Yaskawa INFORM job: SKRZYNIA_4640_0_STOPNI_1OBR.JBI

/JOB
//NAME SKRZYNIA_4640_0_STOPNI_1OBR
///FOLDERNAME 02-SKRZYNIE_JOBS
//POS
///NPOS 503,503,0,43,0,0
///TOOL 0
///POSTYPE PULSE
///PULSE
C00000=1055,-24125,84372,288,19725,204
C00001=1055,-24125,84372,288,19725,204
C00002=0,-15438,65714,0,-68532,0
C00003=25524,-25821,36823,19654,-58495,38520
C00004=23988,-24960,37134,18595,-57837,38812
C00005=22822,-23954,37534,17811,-57199,39017
C00006=22935,-24057,37491,17887,-57262,38997
C00007=20006,-24258,37408,15644,-56932,39751
C00008=24402,-25289,37013,18874,-58060,38740
C00009=22585,-24665,40358,17164,-59622,30036
C00010=23477,-23257,40205,18030,-58646,29630
C00011=22519,-22398,40568,17384,-58125,29795
C00012=22700,-22567,40495,17506,-58225,29764
C00013=19339,-22794,40398,14955,-57865,30607
C00014=24825,-24328,39798,18931,-59350,29401
C00015=25524,-25821,36823,19654,-58495,38520
C00016=23988,-24960,37134,18595,-57837,38812
C00017=22822,-23954,37534,17811,-57199,39017
C00018=22935,-24057,37491,17887,-57262,38997
C00019=20006,-24258,37408,15644,-56932,39751
C00020=24402,-25289,37013,18874,-58060,38740
C00021=22585,-24665,40358,17164,-59622,30036
C00022=23477,-23257,40205,18030,-58646,29630
C00023=22519,-22398,40568,17384,-58125,29795
C00024=22700,-22567,40495,17506,-58225,29764
C00025=19339,-22794,40398,14955,-57865,30607
C00026=24825,-24328,39798,18931,-59350,29401
C00027=32755,-32613,25711,29640,-48730,33694
C00028=25632,-30899,26166,23992,-46203,35378
C00029=24264,-29862,26497,22996,-45413,35639
C00030=24403,-29974,26459,23097,-45496,35612
C00031=20575,-30233,26374,19602,-44891,36810
C00032=26556,-31526,25988,24663,-46720,35206
C00033=31152,-34007,25432,27964,-49085,34371
C00034=14779,-22420,82153,5620,-31515,42478
C00035=14779,-22420,82153,5620,-31515,42478
C00036=27667,-31817,30876,40298,-29340,25942
C00037=30467,-34548,18624,42252,-31099,25545
C00038=27667,-31817,21023,40298,-29340,25942
C00039=26226,-30681,21430,39338,-28403,26129
C00040=26403,-30829,21375,39455,-28520,26106
C00041=23300,-31093,21277,35654,-27590,27434
C00042=27667,-31817,21023,40298,-29340,25942
C00043=33767,-35384,20030,44426,-32984,25136
C00044=17528,-33021,25719,14295,-44761,40001
C00045=28412,-21339,35361,20830,-70681,36412
C00046=27333,-20260,35973,20228,-70115,36596
C00047=27560,-20497,35837,20355,-70235,36556
C00048=24830,-20816,35654,18694,-69859,37222
C00049=28877,-18893,40191,20941,-72149,36569
C00050=27817,-32566,25782,25532,-47502,36865
C00051=25779,-31294,26110,24054,-46400,37243
C00052=24344,-30243,26427,23007,-45578,37515
C00053=24432,-30312,26405,23072,-45630,37498
C00054=20021,-30599,26315,19050,-44944,38872
C00055=26262,-31616,26021,24405,-46667,37153
C00056=27439,-32346,25835,25259,-47302,36935
C00057=25659,-31170,26146,23974,-46312,37260
C00058=24581,-30384,26384,23190,-45695,37464
C00059=24689,-30466,26358,23269,-45758,37444
C00060=20001,-30771,26264,18999,-45026,38899
C00061=26308,-31607,26026,24448,-46671,37139
C00062=26309,-31604,29506,24448,-46670,37138
C00063=58801,-24999,56179,43319,-3155,35712
C00064=58801,-24999,56179,43319,-3155,35712
C00065=58801,-24999,56179,43319,-54497,35712
C00066=29920,-29398,24569,49034,-27892,27689
C00067=29115,-28721,24834,48649,-27358,27707
C00068=27674,-27540,25333,47889,-26423,27783
C00069=27794,-27645,25287,47952,-26502,27777
C00070=24751,-27949,25156,44290,-25406,29014
C00071=29115,-28721,24834,48649,-27358,27707
C00072=40370,-34602,23054,55084,-33911,26929
C00073=27585,-47842,-289,32095,-40789,28095
C00074=4801,-35772,25187,4593,-28023,-82032
C00075=17634,-23800,39238,9573,-31425,-73339
C00076=17634,-23800,39238,9573,-31425,-73339
C00077=16549,-22464,39800,8390,-30730,-72975
C00078=16684,-22641,39722,8536,-30818,-73021
C00079=16684,-19968,45512,8078,-32771,-72767
C00080=17634,-23800,39238,9573,-31425,-73339
C00081=17837,-21535,44509,9322,-33342,-73155
C00082=17837,-21535,44509,9322,-33342,-73155
C00083=16866,-20378,45014,8305,-32755,-72853
C00084=17032,-20588,44918,8481,-32857,-72905
C00085=17032,-17542,51480,8009,-35060,-72636
C00086=17837,-21535,44509,9322,-33342,-73155
C00087=-20829,-18800,50532,-12466,-37179,-77446
C00088=-19934,-17904,50946,-11618,-36715,-77676
C00089=-20044,-18019,50891,-11723,-36773,-77647
C00090=-20044,-15288,56753,-11218,-38713,-77950
C00091=-20966,-18928,50473,-12596,-37250,-77413
C00092=-20884,-26676,33664,-14451,-31668,-76336
C00093=-20884,-26676,33664,-14451,-31668,-76336
C00094=-19557,-25338,34176,-13080,-30873,-76751
C00095=-19691,-25483,34117,-13220,-30955,-76709
C00096=-19691,-22773,39998,-12506,-32911,-77106
C00097=-20642,-26447,33747,-14206,-31526,-76411
C00098=-33629,-40566,17444,-29603,-33447,-71192
C00099=-33629,-40566,17444,42578,-32312,-84654
C00100=-42160,-31266,16400,42578,-32312,-84654
C00101=-87798,-804,48829,-20188,-26072,-60966
C00102=-76454,-11934,10236,-25964,7954,-64922
C00103=-76448,-11928,10235,-25961,7944,-64914
C00104=-68643,-7759,-23318,-14097,50582,-74897
C00105=-70868,-8793,-8075,-29663,30364,-70765
C00106=-67243,-1968,12282,-49553,26687,-63567
C00107=-68655,-309,14069,-48513,25966,-64203
C00108=-67497,-1678,12591,-49367,26558,-63682
C00109=-71436,-723,2905,-26484,35140,-73726
C00110=-71436,176,6426,-27636,33595,-73066
C00111=-71434,778,8668,-28412,32633,-72624
C00112=-68624,-2689,-85,-28291,36551,-72622
C00113=-99375,3692,5712,40719,48607,-84097
C00114=-94964,4957,10918,40408,44640,-83792
C00115=-93063,6047,12199,39572,43744,-83178
C00116=-94964,4957,10918,40408,44640,-83792
C00117=-94964,5754,13918,41385,43553,-84439
C00118=-94964,4957,10918,40408,44640,-83792
C00119=-90271,-412,-5146,23417,46876,-76529
C00120=-83133,-4088,-8267,6704,41492,-71542
C00121=-83133,-4088,-8267,6704,41492,-71542
C00122=-83133,-4088,-8267,6704,41492,-11598
C00123=-83133,-16026,-8267,6704,41492,-11598
C00124=-83133,-16026,-8267,6704,41492,-11598
C00125=-48225,-19387,30619,3889,32460,-6728
C00126=56943,-39861,25115,1795,-37402,-69601
C00127=29960,-38386,-19607,-115769,-41858,-24264
C00128=65721,-6478,18155,-133323,-22195,3361
C00129=70544,4411,32968,-134868,-18623,4660
C00130=71874,8263,38598,-134556,-17327,4659
C00131=72629,9390,40002,-135279,-16924,5107
C00132=71441,7638,37831,-134139,-17555,4406
C00133=77146,8888,25050,-166574,-32612,18372
C00134=77146,10029,28643,-166204,-31014,18167
C00135=77146,11198,32202,-165803,-29459,17947
C00136=75508,4678,16951,-165715,-35157,17778
C00137=68680,12216,24468,-164340,-40455,-13359
C00138=68362,12845,25743,-164045,-40097,-13561
C00139=68362,13700,28585,-163752,-38808,-13742
C00140=68362,12845,25743,-164045,-40097,-13561
C00141=64993,-1168,28876,-102971,-10760,-49875
C00142=63888,481,30670,-102324,-11438,-50313
C00143=64993,-1168,28876,-102971,-10760,-49875
C00144=58588,-14653,4620,-120782,-19611,-35794
C00145=29960,-38386,-19607,-115769,-41858,-24264
C00146=56943,-39861,25115,1795,-37402,-69601
C00147=-1002,-39861,25115,1795,-37402,-69601
C00148=-1001,-39858,25114,1795,-37402,0
C00149=6591,-33902,35532,5956,-1761,-1932
C00150=6592,-33900,35531,103508,-35512,-26314
C00151=-99253,-13690,44082,59847,13407,-31313
C00152=-85045,-36869,-4353,28502,-22832,-52282
C00153=-92346,-18713,13565,21110,-22545,-55257
C00154=-85732,-21202,11427,30682,-24763,-59235
C00155=-84559,-15616,15722,33768,-24118,-60665
C00156=-84150,-13282,17685,34842,-23935,-61163
C00157=-83260,-12880,18034,36130,-24218,-61709
C00158=-84150,-13282,17685,34842,-23935,-61163
C00159=-85365,-11775,19006,33430,-23307,-60600
C00160=-84150,-13282,17685,34842,-23935,-61163
C00161=-85786,-16909,14677,31743,-23900,-59790
C00162=-84150,-13282,17685,34842,-23935,-61163
C00163=-83215,-12861,18051,36194,-24233,-61735
C00164=-84150,-13282,17685,34842,-23935,-61163
C00165=-85327,-11825,18959,33476,-23327,-60618
C00166=-84150,-13282,17685,34842,-23935,-61163
C00167=-87841,-18519,13420,28367,-23534,-58339
C00168=-84150,-13282,17685,34842,-23935,-61163
C00169=-83292,-12894,18020,36083,-24208,-61688
C00170=-84150,-13282,17685,34842,-23935,-61163
C00171=-85185,-12008,18799,33646,-23400,-60687
C00172=-84150,-13282,17685,34842,-23935,-61163
C00173=-86371,-18277,13606,30568,-23951,-59265
C00174=-84345,-13370,17612,34554,-23873,-61041
C00175=-83240,-12871,18042,36158,-24225,-61720
C00176=-84345,-13370,17612,34554,-23873,-61041
C00177=-85365,-12110,18711,33368,-23345,-60568
C00178=-84345,-13370,17612,34554,-23873,-61041
C00179=-86191,-19647,12567,30467,-24278,-59187
C00180=-84345,-13372,17610,34552,-23873,-61039
C00181=-83096,-12807,18098,36363,-24268,-61804
C00182=-84345,-13372,17610,34552,-23873,-61039
C00183=-85268,-12232,18600,33480,-23393,-60612
C00184=-84345,-13372,17610,34552,-23873,-61039
C00185=-84814,-16043,15376,33312,-24093,-60464
C00186=-84104,-13265,17702,34906,-23948,-61189
C00187=-82960,-12743,18153,36555,-24313,-61887
C00188=-84104,-13265,17702,34906,-23948,-61189
C00189=-84979,-12194,18635,33901,-23496,-60788
C00190=-84104,-13265,17702,34906,-23948,-61189
C00191=-86610,-16845,14732,30573,-23614,-59301
C00192=-84104,-13265,17702,34906,-23948,-61189
C00193=-82793,-12667,18222,36790,-24370,-61986
C00194=-84104,-13265,17702,34906,-23948,-61189
C00195=-84888,-12305,18537,34004,-23540,-60830
C00196=-84104,-13265,17702,34906,-23948,-61189
C00197=-83806,-19585,12613,33764,-25080,-60559
C00198=-83675,-13072,17868,35530,-24083,-61453
C00199=-82553,-12556,18319,37130,-24451,-62127
C00200=-83675,-13072,17868,35530,-24083,-61453
C00201=-84378,-12223,18610,34735,-23716,-61138
C00202=-83675,-13072,17868,35530,-24083,-61453
C00203=-87149,-17993,13826,29513,-23647,-58830
C00204=-84104,-13265,17702,34906,-23948,-61189
C00205=-82640,-12594,18285,37014,-24425,-62079
C00206=-84104,-13265,17702,34906,-23948,-61189
C00207=-84792,-12429,18430,34119,-23592,-60877
C00208=-84104,-13265,17702,34906,-23948,-61189
C00209=-83583,-9185,30892,23668,-36042,-57025
C00210=-85789,-8328,35795,20592,-37093,-55378
C00211=-85786,-16735,14816,31782,-23869,-59812
C00212=-84103,-13263,17702,34906,-23947,-61191
C00213=-83225,-12865,18046,36177,-24227,-61729
C00214=-84103,-13263,17702,34906,-23947,-61191
C00215=-84774,-12447,18412,34138,-23599,-60886
C00216=-84103,-13263,17702,34906,-23947,-61191
C00217=-86149,-16246,6730,18897,-35239,-57128
C00218=-86244,-15289,7532,18875,-35060,-57127
C00219=-85361,-14893,7870,19824,-35193,-57574
C00220=-86244,-15289,7532,18875,-35060,-57127
C00221=-86889,-14409,8282,18264,-34784,-56850
C00222=-86244,-15289,7532,18875,-35060,-57127
C00223=-90262,-21765,2389,14114,-35574,-54847
C00224=-90262,-21765,2389,28730,-17672,-54847
C00225=-89967,-19086,25635,28730,-17672,-54847
C00226=568,-24029,84339,168,19981,112
C00227=568,-24677,83015,164,20405,113
C00228=101153,-24598,83176,165,20353,113
C00229=101153,-24598,83176,165,20353,113
C00230=89967,-19086,25635,-28730,-17672,54847
C00231=90262,-21765,2389,-28730,-17672,54847
C00232=86932,-18662,4771,-17876,-35519,56628
C00233=86578,-15436,7408,-18515,-35011,56957
C00234=85428,-14922,7844,-19753,-35183,57541
C00235=84405,-14447,8250,-20842,-35348,58054
C00236=85428,-14922,7844,-19753,-35183,57541
C00237=86134,-13973,8661,-19091,-34881,57237
C00238=85428,-14922,7844,-19753,-35183,57541
C00239=85786,-16735,14816,-31782,-23869,59812
C00240=83514,-12996,17929,-35760,-24132,61552
C00241=82296,-12429,18424,-37488,-24534,62281
C00242=83514,-12996,17929,-35760,-24132,61552
C00243=84266,-12085,18725,-34910,-23738,61214
C00244=83514,-12996,17929,-35760,-24132,61552
C00245=87323,-6914,39851,-18853,-38149,44508
C00246=83118,-12818,18089,-36330,-24263,61791
C00247=81969,-12276,18566,-37944,-24648,62472
C00248=83118,-12818,18089,-36330,-24263,61791
C00249=83927,-11846,18941,-35423,-23842,61433
C00250=83118,-12818,18089,-36330,-24263,61791
C00251=83806,-19585,12613,-33764,-25080,60559
C00252=83148,-12832,18077,-36287,-24254,61773
C00253=81889,-12236,18598,-38058,-24676,62520
C00254=83148,-12832,18077,-36287,-24254,61773
C00255=83900,-11930,18867,-35446,-23862,61440
C00256=83148,-12832,18077,-36287,-24254,61773
C00257=86610,-16845,14732,-30573,-23614,59301
C00258=82493,-13239,17725,-37070,-24559,62089
C00259=81442,-12739,18159,-38529,-24915,62703
C00260=82493,-13239,17725,-37070,-24559,62089
C00261=83435,-12133,18689,-36040,-24063,61682
C00262=82493,-13239,17725,-37070,-24559,62089
C00263=84814,-16043,15376,-33312,-24093,60464
C00264=82555,-13613,17404,-36910,-24580,62015
C00265=81369,-13053,17885,-38558,-24979,62709
C00266=82555,-13613,17404,-36910,-24580,62015
C00267=83568,-12431,18429,-35805,-24046,61580
C00268=82555,-13613,17404,-36910,-24580,62015
C00269=86191,-19647,12567,-30467,-24278,59187
C00270=82500,-13648,17375,-36975,-24607,62039
C00271=81594,-13224,17740,-38236,-24911,62571
C00272=82500,-13648,17375,-36975,-24607,62039
C00273=83449,-12543,18332,-35941,-24104,61633
C00274=82500,-13648,17375,-36975,-24607,62039
C00275=86371,-18277,13606,-30568,-23951,59265
C00276=82904,-13790,17251,-36416,-24470,61808
C00277=81796,-13275,17692,-37971,-24838,62464
C00278=82904,-13790,17251,-36416,-24470,61808
C00279=83696,-12867,18046,-35547,-24051,61466
C00280=82904,-13790,17251,-36416,-24470,61808
C00281=87841,-18519,13420,-28367,-23534,58339
C00282=82748,-13879,17174,-36603,-24542,61883
C00283=81789,-13434,17554,-37946,-24861,62449
C00284=82748,-13879,17174,-36603,-24542,61883
C00285=83603,-12888,18026,-35668,-24086,61514
C00286=82748,-13879,17174,-36603,-24542,61883
C00287=85786,-16909,14677,-31743,-23900,59790
C00288=82339,-14116,16972,-37087,-24733,62079
C00289=81557,-13752,17280,-38171,-24994,62536
C00290=82339,-14116,16972,-37087,-24733,62079
C00291=83390,-12909,18006,-35951,-24172,61633
C00292=82339,-14116,16972,-37087,-24733,62079
C00293=85732,-21202,11427,-30682,-24763,59235
C00294=82398,-14365,16763,-36952,-24745,62014
C00295=81340,-13876,17176,-38416,-25096,62632
C00296=82398,-14365,16763,-36952,-24745,62014
C00297=83629,-12951,17972,-35620,-24090,61491
C00298=82398,-14365,16763,-36952,-24745,62014
C00299=83775,-36460,5778,-32556,-23750,56951
C00300=69856,-53931,-13446,-33557,-28911,29591
C00301=43695,-41610,22646,45477,-37580,9181
C00302=79833,-32060,29151,65065,-75499,17030
C00303=46589,-23543,32575,47437,-59456,19719
C00304=35046,-28601,21000,31995,-60106,26294
C00305=20995,-31929,9410,15929,-60729,34224
C00306=58029,-25484,23838,55879,-68285,17494
C00307=64424,-28491,31029,58630,-66351,17656
C00308=34280,-39622,35434,31197,-32089,9395
C00309=0,-52280,40443,0,6876,0
C00310=23755,-47704,18289,26329,-25233,13971
C00311=32804,-46073,6525,41905,-31120,14425
C00312=62562,-39100,6547,70046,-55853,12125
C00313=48126,-33841,8393,64372,-47199,12361
C00314=31253,-44096,-7366,36514,-42480,22085
C00315=59828,-44646,-5405,72855,-48572,12139
C00316=0,-38761,66314,0,-763,0
C00317=0,-44757,54667,0,2744,0
C00318=16657,-42063,37160,20008,-15173,6616
C00319=40382,-38226,12225,48505,-40693,16039
C00320=55481,-27484,23768,62968,-54833,11978
C00321=49931,-26522,24223,59987,-51967,12537
C00322=41382,-34078,10932,46059,-50502,16311
C00323=55330,-33748,11238,57660,-59334,12681
C00324=57521,-31202,17284,65112,-55174,10876
C00325=49952,-26929,23567,59763,-52208,12588
C00326=49645,-31441,12217,55064,-56016,13120
C00327=55330,-33748,11238,57660,-59334,12681
C00328=78664,-24436,10378,82837,-79111,12029
C00329=75189,-23065,11287,81851,-76948,11927
C00330=75189,-45249,11287,81851,-38847,11927
C00331=39199,-45249,11287,81851,-83130,11927
C00332=39199,-45249,11287,81851,-83130,11927
C00333=0,-24026,84338,1,19977,2
C00334=0,-24026,84338,1,19977,2
C00335=4264,-34194,25387,4006,-26954,-29436
C00336=4264,-34194,25387,4006,-26954,-81856
C00337=-21478,-27798,32214,-15234,-31599,-76056
C00338=-19679,-23059,39354,-12567,-32689,-77067
C00339=16724,-20576,44291,8212,-32395,-72836
C00340=21329,-26386,39716,13285,-34016,-74401
C00341=-23778,-26243,38799,-16502,-35132,-75964
C00342=-20075,-15782,55752,-11329,-38404,-77896
C00343=16874,-17447,51356,7863,-34895,-72604
C00344=18580,-28601,30698,11472,-29284,-74138
C00345=6126,-41331,18955,6697,-26557,-30383
C00346=1,-24024,84337,2,19973,1
C00347=-64243,-26178,31107,-39513,40312,-5844
C00348=-72148,3973,56008,-35470,42045,-10522
C00349=-72090,16396,76301,-42067,35650,-6519
C00350=-69388,15725,61378,-31740,35177,-8719
C00351=-69127,27099,75569,-32744,34250,-8088
C00352=-67573,2495,11285,-21767,57629,-15193
C00353=-77819,19629,29798,-10454,63174,-20704
C00354=-72990,23583,14304,-10735,77209,-20379
C00355=-74593,38003,46707,-11043,65751,-19814
C00356=-73236,38943,48295,-11400,65557,-19316
C00357=-73329,42107,51779,-6346,67443,-19636
C00358=-87142,34654,46174,17622,63862,-25393
C00359=-87240,36727,48611,18897,66604,-25032
C00360=-99033,21517,12213,24947,79702,-26203
C00361=-91500,-14196,-34781,24472,81625,-22832
C00362=-100472,-45007,-27818,8167,67201,-29302
C00363=0,-36642,16905,0,48372,0
C00364=66009,-61997,-62105,21406,63483,18379
C00365=97242,-23579,-39442,10179,68876,30321
C00366=73684,-7073,-17511,24638,68131,29022
C00367=59136,7235,6676,33270,66602,27507
C00368=54816,14937,6234,39741,69494,31070
C00369=54365,20668,19279,41017,66202,29418
C00370=64503,4223,2857,29650,48528,26647
C00371=75622,3202,-3149,3890,49494,34281
C00372=88036,13177,2413,-18568,66573,35876
C00373=90462,21593,10123,-22613,76266,34479
C00374=92450,29224,20002,-25750,81642,33727
C00375=94949,8131,-12163,-20291,74229,36861
C00376=94949,8084,-13484,-20215,75047,36712
C00377=70412,-34016,-52305,-11724,65624,29757
C00378=44268,-30306,-1568,-7370,48673,18708
C00379=1,-24024,84337,2,19973,1
C00380=1,-24024,84337,2,19973,1
C00381=35720,-26719,45333,36814,-39824,4350
C00382=31427,-24257,37066,30413,-51503,29688
C00383=34144,-17362,32181,27785,-74498,33370
C00384=48608,-25286,29226,41890,-68866,29453
C00385=62093,-26534,55494,45669,-73540,27410
C00386=1,-24024,84337,2,19973,1
C00387=39943,-41903,29008,37348,-30478,1122
C00388=50712,-45163,3694,54202,-48634,13777
C00389=34255,-38662,5079,45062,-39023,15547
C00390=40870,-40863,-13430,41877,-55633,22482
C00391=59329,-52422,-25741,69939,-52774,12149
C00392=61512,-31790,21528,108331,-82342,18812
C00393=13547,-32557,41617,75619,-64512,89
C00394=-91085,-34291,10385,1908,-24348,-42097
C00395=-86191,-19647,12567,30467,-24278,-59187
C00396=-99336,-11722,19052,-14323,-20229,-40037
C00397=-98356,-11562,19564,-10422,-20330,-41507
C00398=-99474,-20389,12397,-11593,-22150,-41069
C00399=0,-52280,40443,0,6876,0
C00400=98750,-34911,19055,13387,-20552,33529
C00401=85481,-22689,10385,-30594,-25183,59147
C00402=97204,-12655,18233,8807,-19987,42423
C00403=97248,-12883,18033,8874,-20029,42393
C00404=96230,-24528,9149,6144,-22576,43630
C00405=0,-52280,40443,0,6876,0
C00406=0,-52280,40443,0,6876,0
C00407=-90140,-60305,18108,-2708,1721,-7625
C00408=-95594,-27428,6866,-4663,-19832,-42154
C00409=-99356,-13410,18355,-15385,-17730,-37479
C00410=-99591,-10931,20459,-16242,-17374,-37088
C00411=-99412,-10883,20509,-15863,-17339,-37249
C00412=-100555,-16348,15834,-17428,-18409,-36628
C00413=-90140,-60305,18108,-2708,1721,-7625
C00414=0,-52280,40443,0,6876,0
C00415=84259,-57935,27522,-3761,3673,6310
C00416=86507,-39672,4297,-27618,-16640,46340
C00417=79502,-31038,5321,-35142,-29552,60614
C00418=87509,-17632,14108,-29072,-23467,58651
C00419=100494,-12641,18246,19637,-20925,37756
C00420=99867,-15453,10402,24266,-14765,33998
C00421=100699,-20865,6123,24471,-16015,33991
C00422=86507,-39672,4297,-27618,-16640,46340
C00423=84259,-57935,27522,-3761,3673,6310
C00424=0,-52280,40443,0,6876,0
C00425=0,-27933,77061,0,20812,0
C00426=0,-27933,77061,0,20812,0
C00427=0,-52280,40443,0,6876,0
C00428=-91970,-60791,14435,-3343,512,-9412
C00429=-99196,-15868,16098,-13748,-19297,-38710
C00430=-99196,-15868,16098,-13748,-19297,-38710
C00431=-99196,-15868,16098,-13748,-19297,-38710
C00432=-85896,-11794,19566,31613,-21074,-58206
C00433=-87494,-11929,19445,26784,-20178,-56163
C00434=-99562,-16264,15781,-14410,-19427,-38431
C00435=-99196,-15868,16098,-13748,-19297,-38710
C00436=-91970,-60791,14435,-3343,512,-9412
C00437=0,-52280,40443,0,6876,0
C00438=91083,-60784,14823,-9043,-825,15173
C00439=83869,-19403,12921,-33769,-24740,60260
C00440=83869,-19403,12921,-33769,-24740,60260
C00441=83420,-14897,16486,-35538,-24144,61113
C00442=90681,-11839,19658,-13770,-20778,51433
C00443=90505,-11641,19895,-14005,-20849,51502
C00444=95871,-14889,15992,4901,-19605,43825
C00445=83869,-19403,12921,-33769,-24740,60260
C00446=91083,-60784,14823,-9043,-825,15173
C00447=0,-52280,40443,0,6876,0
C00448=-91526,-60598,16699,7584,176,-13289
C00449=-94392,-6553,48683,5805,-47321,-49764
C00450=-88951,-345,54953,10686,-47392,-51569
C00451=-88305,5764,62037,11205,-47732,-51744
C00452=-91201,-14114,9416,8552,-34389,-51801
C00453=-84917,-15593,15742,33275,-23984,-60461
C00454=-81669,-15982,15425,37506,-25258,-62202
C00455=-79867,-25377,9541,37586,-25936,-59971
C00456=-91415,-60262,16631,7870,-73,-13734
C00457=24,-24029,84339,7,19981,5
C00458=160,-24029,84339,47,19981,32
C00459=99096,-24029,84339,47,19981,32
C00460=99096,-24029,84339,47,19981,32
C00461=89967,-19086,25635,-28730,-17672,54847
C00462=85786,-16735,14816,-31782,-23869,59812
C00463=83492,-14473,16674,-35480,-24338,61406
C00464=82747,-11488,19289,-37317,-24361,62210
C00465=85506,-13730,8787,-19466,-34817,57474
C00466=85505,-16299,6686,-19564,-35388,57437
C00467=89967,-19086,25635,-28730,-17672,54847
C00468=568,-24029,84339,168,19981,112
C00469=568,-24029,84339,168,19981,112
C00470=-91970,-60791,14435,-3343,512,-9412
C00471=-86948,-23217,10819,28314,-23349,-56438
C00472=-85895,-16522,15767,31843,-22281,-58087
C00473=-93744,1669,52928,2829,-38206,-34736
C00474=-93484,-766,47198,3260,-36104,-34933
C00475=-86145,-24679,9854,29028,-23971,-56682
C00476=-100471,-58311,4157,14142,-4822,-27614
C00477=-68517,-58311,4157,14142,-4822,-27614
C00478=0,-52280,40443,0,6876,0
C00479=91083,-60784,14823,-9043,-825,15173
C00480=83869,-19403,12921,-33769,-24740,60260
C00481=82620,-18743,14708,-32942,-26226,58979
C00482=84031,-4887,35984,-19530,-40379,54984
C00483=84316,-7987,27276,-19995,-38113,55712
C00484=84798,-22668,11879,-29033,-26372,57255
C00485=91083,-60784,14823,-9043,-825,15173
C00486=0,-52280,40443,0,6876,0
C00487=-100896,-36216,1995,-16119,-20751,-34692
C00488=-97287,-29142,12714,-8673,-22288,-37832
C00489=-86191,-19647,12567,30467,-24278,-59187
C00490=-85671,-16302,15857,30808,-24404,-58999
C00491=-100216,-10426,22391,-15020,-22581,-38655
C00492=-96259,-10424,22189,-2878,-17380,-43087
C00493=-87910,-17792,15835,25414,-24996,-56048
C00494=-97287,-29142,12714,-8673,-22288,-37832
C00495=0,-47400,49619,0,4231,0
C00496=92301,-25634,22749,2368,-15645,37646
C00497=83738,-18329,13570,-34202,-24868,60772
C00498=90255,-12942,18284,-15153,-20833,52586
C00499=93508,-13158,18002,-4292,-20124,47959
C00500=79675,-24852,9157,-38810,-28565,62243
C00501=91863,-41556,2664,1531,-13798,37970
C00502=0,-46824,50714,0,3911,0
BC00000=413138
BC00001=413138
BC00002=413138
BC00003=290246
BC00004=290246
BC00005=290246
BC00006=290246
BC00007=290246
BC00008=290246
BC00009=347127
BC00010=347132
BC00011=347132
BC00012=347132
BC00013=347132
BC00014=347132
BC00015=413134
BC00016=413134
BC00017=413134
BC00018=413134
BC00019=413134
BC00020=413134
BC00021=474623
BC00022=474628
BC00023=474628
BC00024=474628
BC00025=474628
BC00026=474628
BC00027=522849
BC00028=522849
BC00029=522849
BC00030=522849
BC00031=522849
BC00032=522849
BC00033=522849
BC00034=431251
BC00035=493719
BC00036=553627
BC00037=550624
BC00038=553627
BC00039=553627
BC00040=553627
BC00041=553627
BC00042=553627
BC00043=553627
BC00044=686969
BC00045=712250
BC00046=712250
BC00047=712250
BC00048=712250
BC00049=712250
BC00050=708270
BC00051=708270
BC00052=708270
BC00053=708270
BC00054=708270
BC00055=708270
BC00056=754823
BC00057=754823
BC00058=754823
BC00059=754823
BC00060=754823
BC00061=754823
BC00062=733905
BC00063=652761
BC00064=769869
BC00065=769869
BC00066=788736
BC00067=788736
BC00068=788736
BC00069=788736
BC00070=788736
BC00071=788736
BC00072=788736
BC00073=888392
BC00074=834347
BC00075=849708
BC00076=849708
BC00077=849708
BC00078=849708
BC00079=849708
BC00080=849708
BC00081=854154
BC00082=854154
BC00083=854154
BC00084=854154
BC00085=854154
BC00086=854154
BC00087=854154
BC00088=854154
BC00089=854154
BC00090=854154
BC00091=854154
BC00092=854154
BC00093=854154
BC00094=854154
BC00095=854154
BC00096=854154
BC00097=854154
BC00098=854154
BC00099=854154
BC00100=854154
BC00101=854154
BC00102=854154
BC00103=871906
BC00104=882992
BC00105=899696
BC00106=899696
BC00107=899696
BC00108=899696
BC00109=899696
BC00110=899696
BC00111=899697
BC00112=899697
BC00113=899697
BC00114=899697
BC00115=899697
BC00116=899697
BC00117=899697
BC00118=899697
BC00119=890074
BC00120=875440
BC00121=850175
BC00122=850175
BC00123=850175
BC00124=816993
BC00125=782560
BC00126=854154
BC00127=854154
BC00128=854154
BC00129=870368
BC00130=875529
BC00131=875529
BC00132=875529
BC00133=875529
BC00134=875529
BC00135=875529
BC00136=875529
BC00137=875529
BC00138=875529
BC00139=875529
BC00140=875529
BC00141=875529
BC00142=875529
BC00143=875529
BC00144=870016
BC00145=823432
BC00146=792710
BC00147=792710
BC00148=854156
BC00149=785093
BC00150=785096
BC00151=785096
BC00152=854699
BC00153=886829
BC00154=902188
BC00155=902188
BC00156=902188
BC00157=902188
BC00158=902188
BC00159=902188
BC00160=902188
BC00161=840744
BC00162=840744
BC00163=840744
BC00164=840744
BC00165=840744
BC00166=840744
BC00167=779300
BC00168=779300
BC00169=779300
BC00170=779300
BC00171=779300
BC00172=779300
BC00173=717855
BC00174=717855
BC00175=717855
BC00176=717855
BC00177=717855
BC00178=717855
BC00179=656405
BC00180=656405
BC00181=656405
BC00182=656405
BC00183=656405
BC00184=656405
BC00185=594961
BC00186=594961
BC00187=594961
BC00188=594961
BC00189=594961
BC00190=594961
BC00191=533517
BC00192=533517
BC00193=533517
BC00194=533517
BC00195=533517
BC00196=533517
BC00197=472073
BC00198=472073
BC00199=472073
BC00200=472073
BC00201=472073
BC00202=472073
BC00203=410629
BC00204=410629
BC00205=410629
BC00206=410629
BC00207=410629
BC00208=410629
BC00209=410629
BC00210=349186
BC00211=349186
BC00212=349186
BC00213=349186
BC00214=349186
BC00215=349186
BC00216=349186
BC00217=336469
BC00218=336469
BC00219=336469
BC00220=336469
BC00221=336469
BC00222=336469
BC00223=336469
BC00224=336469
BC00225=336469
BC00226=336469
BC00227=511557
BC00228=512005
BC00229=363797
BC00230=336469
BC00231=336469
BC00232=337415
BC00233=337415
BC00234=337415
BC00235=337415
BC00236=337415
BC00237=337415
BC00238=337415
BC00239=349186
BC00240=350137
BC00241=350137
BC00242=350137
BC00243=350137
BC00244=350137
BC00245=410629
BC00246=411580
BC00247=411580
BC00248=411580
BC00249=411580
BC00250=411580
BC00251=472073
BC00252=473025
BC00253=473025
BC00254=473025
BC00255=473025
BC00256=473025
BC00257=533517
BC00258=534468
BC00259=534468
BC00260=534468
BC00261=534468
BC00262=534468
BC00263=594961
BC00264=594961
BC00265=594961
BC00266=594961
BC00267=594961
BC00268=594961
BC00269=656405
BC00270=657350
BC00271=657350
BC00272=657350
BC00273=657350
BC00274=657350
BC00275=717855
BC00276=718799
BC00277=718799
BC00278=718799
BC00279=718799
BC00280=718799
BC00281=779300
BC00282=780245
BC00283=780245
BC00284=780245
BC00285=780245
BC00286=780245
BC00287=840744
BC00288=841691
BC00289=841691
BC00290=841691
BC00291=841691
BC00292=841691
BC00293=902188
BC00294=903136
BC00295=903136
BC00296=903136
BC00297=903136
BC00298=903136
BC00299=866428
BC00300=742376
BC00301=723595
BC00302=717171
BC00303=717171
BC00304=716481
BC00305=715784
BC00306=716000
BC00307=727625
BC00308=662842
BC00309=820009
BC00310=882789
BC00311=908954
BC00312=917484
BC00313=934308
BC00314=923719
BC00315=887066
BC00316=801718
BC00317=477813
BC00318=443512
BC00319=475338
BC00320=456696
BC00321=456696
BC00322=417276
BC00323=417276
BC00324=333808
BC00325=332068
BC00326=295166
BC00327=294388
BC00328=493986
BC00329=514306
BC00330=485368
BC00331=485368
BC00332=586924
BC00333=635329
BC00334=727981
BC00335=816098
BC00336=821314
BC00337=854154
BC00338=854154
BC00339=849707
BC00340=843941
BC00341=839452
BC00342=854154
BC00343=854154
BC00344=853382
BC00345=856974
BC00346=704835
BC00347=720197
BC00348=720197
BC00349=776907
BC00350=796793
BC00351=821732
BC00352=853664
BC00353=853664
BC00354=881173
BC00355=881173
BC00356=881173
BC00357=881174
BC00358=881174
BC00359=881175
BC00360=881175
BC00361=881175
BC00362=795833
BC00363=754431
BC00364=837971
BC00365=877091
BC00366=877092
BC00367=877092
BC00368=907339
BC00369=907339
BC00370=907339
BC00371=907339
BC00372=907339
BC00373=907342
BC00374=907342
BC00375=907342
BC00376=880936
BC00377=880936
BC00378=812123
BC00379=689474
BC00380=565631
BC00381=569135
BC00382=579756
BC00383=579756
BC00384=579756
BC00385=586542
BC00386=728933
BC00387=790967
BC00388=835726
BC00389=835726
BC00390=835726
BC00391=835752
BC00392=835752
BC00393=704157
BC00394=707357
BC00395=656405
BC00396=656405
BC00397=717855
BC00398=717855
BC00399=637115
BC00400=662303
BC00401=657350
BC00402=657350
BC00403=718803
BC00404=718803
BC00405=633287
BC00406=792672
BC00407=792672
BC00408=896850
BC00409=895720
BC00410=895720
BC00411=925351
BC00412=927080
BC00413=792672
BC00414=792672
BC00415=792672
BC00416=887446
BC00417=903126
BC00418=903126
BC00419=903126
BC00420=936389
BC00421=936389
BC00422=887446
BC00423=792672
BC00424=792672
BC00425=700249
BC00426=546214
BC00427=546214
BC00428=546211
BC00429=546211
BC00430=406776
BC00431=406776
BC00432=406778
BC00433=468200
BC00434=468200
BC00435=546211
BC00436=546211
BC00437=546214
BC00438=546214
BC00439=507604
BC00440=410782
BC00441=410782
BC00442=410782
BC00443=472720
BC00444=472720
BC00445=507604
BC00446=546214
BC00447=546214
BC00448=516757
BC00449=383716
BC00450=349186
BC00451=349186
BC00452=336469
BC00453=349186
BC00454=410629
BC00455=416512
BC00456=515801
BC00457=520018
BC00458=474013
BC00459=474013
BC00460=403108
BC00461=336469
BC00462=349186
BC00463=349186
BC00464=349186
BC00465=337415
BC00466=337415
BC00467=336469
BC00468=336469
BC00469=428401
BC00470=546211
BC00471=591088
BC00472=591088
BC00473=591088
BC00474=531116
BC00475=529640
BC00476=529640
BC00477=529640
BC00478=529640
BC00479=546214
BC00480=589919
BC00481=595627
BC00482=609761
BC00483=555903
BC00484=534177
BC00485=546214
BC00486=529640
BC00487=765890
BC00488=765890
BC00489=777968
BC00490=778453
BC00491=779252
BC00492=832733
BC00493=840748
BC00494=730002
BC00495=613681
BC00496=714120
BC00497=780224
BC00498=780222
BC00499=841743
BC00500=841743
BC00501=719906
BC00502=630890
///POSTYPE BASE
///RECTAN
///RCONF 1,0,0,0,0,0,0,0,0,0,0,0,0,0,0,0,0,0,0,0,0,0,0,0
P00006=0.000,0.000,0.000,0.0000,0.0000,0.0000
///RCONF 0,0,0,0,0,0,0,0,0,0,0,0,0,0,0,0,0,0,0,0,0,0,0,0
P00021=6.550,-0.003,-5.735,0.0000,0.0000,0.0000
P00022=5.943,-0.018,-6.388,0.0000,0.0000,0.0000
P00023=7.025,-0.019,-7.168,0.0000,0.0000,0.0000
P00024=5.926,-0.047,-4.777,0.0000,0.0000,0.0000
///RCONF 1,0,0,0,0,0,0,0,0,0,0,0,0,0,0,0,0,0,0,0,0,0,0,0
P00098=-0.089,-2.467,4.059,0.0000,0.0000,0.0000
P00099=0.011,-2.380,1.226,0.0000,0.0000,0.0000
P00100=-0.081,2.558,4.482,0.0000,0.0000,0.0000
P00101=0.030,-2.286,2.993,0.0000,0.0000,0.0000
P00102=-0.005,-1.108,1.644,0.0000,0.0000,0.0000
P00103=-0.094,-3.400,4.200,0.0000,0.0000,0.0000
P00104=0.043,-2.127,5.826,0.0000,0.0000,0.0000
P00105=-0.043,0.662,5.286,0.0000,0.0000,0.0000
P00106=-0.018,-2.519,0.237,0.0000,0.0000,0.0000
P00107=-0.008,-4.537,-4.500,0.0000,0.0000,0.0000
P00108=0.014,-3.040,2.637,0.0000,0.0000,0.0000
P00109=0.017,-3.622,2.341,0.0000,0.0000,0.0000
///RCONF 0,0,0,0,0,0,0,0,0,0,0,0,0,0,0,0,0,0,0,0,0,0,0,0
P00280=-0.761,-1.221,0.004,0.0000,0.0000,0.0000
///RCONF 1,0,0,0,0,0,0,0,0,0,0,0,0,0,0,0,0,0,0,0,0,0,0,0
P00281=-0.866,-3.587,-0.008,0.0000,0.0000,0.0000
///RCONF 0,0,0,0,1,0,0,0,0,0,0,0,0,0,0,0,0,0,0,0,0,0,0,0
P00290=-0.023,-0.050,5.560,0.0000,0.0000,0.0000
///RCONF 1,0,0,0,0,0,0,0,0,0,0,0,0,0,0,0,0,0,0,0,0,0,0,0
P00291=0.002,-0.893,4.526,0.0000,0.0000,0.0000
P00301=0.046,-2.112,7.779,0.0000,0.0000,0.0000
P00302=-0.180,-2.409,6.326,0.0000,0.0000,0.0000
///RCONF 0,0,0,0,0,0,0,0,0,0,0,0,0,0,0,0,0,0,0,0,0,0,0,0
P00303=-0.004,-1.437,-4.584,0.0000,0.0000,0.0000
P00304=0.028,-1.666,-4.234,0.0000,0.0000,0.0000
P00305=-0.003,-1.920,-3.501,0.0000,0.0000,0.0000
P00306=0.015,-2.252,-3.054,0.0000,0.0000,0.0000
P00307=0.019,-2.151,-5.077,0.0000,0.0000,0.0000
P00308=-0.003,-2.092,-4.888,0.0000,0.0000,0.0000
P00309=-0.040,-2.205,-4.992,0.0000,0.0000,0.0000
P00310=-0.006,-2.490,-5.925,0.0000,0.0000,0.0000
P00311=-0.007,-2.079,-5.307,0.0000,0.0000,0.0000
P00350=11.519,-0.008,1.149,0.0000,0.0000,0.0000
P00351=13.563,-0.027,-0.653,0.0000,0.0000,0.0000
P00352=13.252,-0.027,-0.827,0.0000,0.0000,0.0000
P00353=10.971,-0.082,0.776,0.0000,0.0000,0.0000
P00354=-0.024,2.508,-1.824,0.0000,0.0000,0.0000
P00355=-0.001,2.528,-1.131,0.0000,0.0000,0.0000
P00356=-0.034,2.921,-0.262,0.0000,0.0000,0.0000
P00357=0.003,3.386,-0.091,0.0000,0.0000,0.0000
P00358=0.014,3.037,-0.020,0.0000,0.0000,0.0000
P00359=-0.005,2.731,0.912,0.0000,0.0000,0.0000
P00360=-0.011,3.412,0.438,0.0000,0.0000,0.0000
//INST
///DATE 2025/06/03 07:49
///ATTR SC,RW
///GROUP1 RB1,BS1
NOP
CALL JOB:MOVE_INTO_TUNNEL
MOVJ C00000 BC00000 VJ=30.00
'------------------------
'------------------------
'SPOINA SRODEK DOL
'------------------------
'------------------------
'POMIAR DO WYJ!! PRZEROBIC NA STD
MOVJ C00001 BC00001 VJ=40.00
MOVJ C00002 BC00002 VJ=40.00
'SPOINA_PODLOGA_BRAK_ROZP
MOVJ C00003 BC00003 VJ=20.00 PL=0
MOVL C00004 BC00004 V=166.7 PL=0
REFP 3 C00005 BC00005
CALL JOB:SEARCH-R1
SET P0098 P0006
SFTON P0098
MOVL C00006 BC00006 V=66.7 PL=0
REFP 3 C00007 BC00007
CALL JOB:SEARCH-R1
SET P0098 P0006
SFTON P0098
MOVL C00008 BC00008 V=333.3 PL=0
SFTOF
'W3L
MOVL C00009 BC00009 V=666.7
MOVL C00010 BC00010 V=166.7 PL=0
REFP 3 C00011 BC00011
CALL JOB:SEARCH-R1
SET P0099 P0006
SFTON P0099
MOVL C00012 BC00012 V=166.7 PL=0
REFP 3 C00013 BC00013
CALL JOB:SEARCH-R1
SET P0099 P0006
SFTON P0099
MOVL C00014 BC00014 V=333.3 PL=0
SFTOF
'SPOINA_PODLOGA_BRAK_ROZP
'W3P
MOVJ C00015 BC00015 VJ=20.00 PL=0
MOVL C00016 BC00016 V=166.7 PL=0
REFP 3 C00017 BC00017
CALL JOB:SEARCH-R1
SET P0100 P0006
SFTON P0100
MOVL C00018 BC00018 V=66.7 PL=0
REFP 3 C00019 BC00019
CALL JOB:SEARCH-R1
SET P0100 P0006
SFTON P0100
MOVL C00020 BC00020 V=333.3 PL=0
SFTOF
'W3L
MOVL C00021 BC00021 V=666.7
MOVL C00022 BC00022 V=166.7 PL=0
REFP 3 C00023 BC00023
CALL JOB:SEARCH-R1
SET P0101 P0006
SFTON P0101
MOVL C00024 BC00024 V=166.7 PL=0
REFP 3 C00025 BC00025
CALL JOB:SEARCH-R1
SET P0101 P0006
SFTON P0101
MOVL C00026 BC00026 V=333.3 PL=0
SFTOF
'W9P
MOVL C00027 BC00027 V=666.7
MOVL C00028 BC00028 V=166.7
REFP 3 C00029 BC00029
CALL JOB:SEARCH-R1
SET P0102 P0006
SFTON P0102
MOVL C00030 BC00030 V=166.7 PL=0
REFP 3 C00031 BC00031
CALL JOB:SEARCH-R1
SET P0102 P0006
SFTON P0102
SFTOF
MOVL C00032 BC00032 V=333.3 PL=0
MOVJ C00033 BC00033 VJ=30.00
MOVJ C00034 BC00034 VJ=30.00
MOVJ C00035 BC00035 VJ=30.00
MOVJ C00036 BC00036 VJ=30.00
'W9L
MOVL C00037 BC00037 V=666.7
MOVL C00038 BC00038 V=166.7
REFP 3 C00039 BC00039
CALL JOB:SEARCH-R1
SET P0103 P0006
SFTON P0103
MOVL C00040 BC00040 V=166.7 PL=0
REFP 3 C00041 BC00041
CALL JOB:SEARCH-R1
SET P0103 P0006
SFTON P0103
MOVL C00042 BC00042 V=333.3 PL=0
SFTOF
MOVJ C00043 BC00043 VJ=30.00
'PRZEJAZ NAD BELKA
'W1P
SFTOF
MOVJ C00044 BC00044 VJ=20.00 PL=0
MOVL C00045 BC00045 V=166.7 PL=0
REFP 3 C00046 BC00046
CALL JOB:SEARCH-R1
SET P0104 P0006
SFTON P0104
MOVL C00047 BC00047 V=166.7 PL=0
REFP 3 C00048 BC00048
CALL JOB:SEARCH-R1
SET P0104 P0006
SFTON P0104
MOVL C00049 BC00049 V=333.3 PL=0
SFTOF
'W1L
MOVL C00050 BC00050 V=666.7
MOVL C00051 BC00051 V=166.7 PL=0
REFP 3 C00052 BC00052
CALL JOB:SEARCH-R1
SET P0105 P0006
SFTON P0105
MOVL C00053 BC00053 V=166.7 PL=0
REFP 3 C00054 BC00054
CALL JOB:SEARCH-R1
SET P0105 P0006
SFTON P0105
MOVL C00055 BC00055 V=333.3 PL=0
SFTOF
MOVL C00056 BC00056 V=666.7
'W10P
MOVL C00057 BC00057 V=166.7 PL=0
REFP 3 C00058 BC00058
CALL JOB:SEARCH-R1
SET P0106 P0006
SFTON P0106
MOVL C00059 BC00059 V=166.7 PL=0
REFP 3 C00060 BC00060
CALL JOB:SEARCH-R1
SET P0106 P0006
SFTON P0106
MOVL C00061 BC00061 V=333.3 PL=0
SFTOF
'W10L
MOVJ C00062 BC00062 VJ=30.00
MOVJ C00063 BC00063 VJ=30.00
MOVJ C00064 BC00064 VJ=30.00
MOVJ C00065 BC00065 VJ=30.00
MOVL C00066 BC00066 V=333.3
MOVL C00067 BC00067 V=166.7 PL=0
REFP 3 C00068 BC00068
CALL JOB:SEARCH-R1
SET P0107 P0006
SFTON P0107
MOVL C00069 BC00069 V=166.7 PL=0
REFP 3 C00070 BC00070
CALL JOB:SEARCH-R1
SET P0107 P0006
SFTON P0107
MOVL C00071 BC00071 V=333.3 PL=0
SFTOF
MOVJ C00072 BC00072 VJ=30.00
'PRZEJAZD
'POMIAR DO WYJ!! PRZEROBIC NA STD
'KONIEC
MOVJ C00073 BC00073 VJ=25.00
MOVJ C00074 BC00074 VJ=50.00
'W5L
MOVJ C00075 BC00075 VJ=30.00 PL=0
MOVL C00076 BC00076 V=166.7
REFP 3 C00077 BC00077
CALL JOB:SEARCH-R1
SET P0021 P0006
SFTON P0021
MOVL C00078 BC00078 V=166.7
REFP 3 C00079 BC00079
CALL JOB:SEARCH-R1
SET P0021 P0006
SFTON P0021
SFTOF
MOVL C00080 BC00080 V=166.7
'W6L
MOVJ C00081 BC00081 VJ=20.00 PL=0
MOVL C00082 BC00082 V=166.7
REFP 3 C00083 BC00083
CALL JOB:SEARCH-R1
SET P0022 P0006
SFTON P0022
MOVL C00084 BC00084 V=166.7
REFP 3 C00085 BC00085
CALL JOB:SEARCH-R1
SET P0022 P0006
SFTON P0022
SFTOF
MOVL C00086 BC00086 V=166.7
'W6P
MOVL C00087 BC00087 V=333.3 PL=0
REFP 3 C00088 BC00088
CALL JOB:SEARCH-R1
SET P0023 P0006
SFTON P0023
MOVL C00089 BC00089 V=166.7
REFP 3 C00090 BC00090
CALL JOB:SEARCH-R1
SET P0023 P0006
SFTON P0023
SFTOF
MOVL C00091 BC00091 V=166.7
'W5P
MOVJ C00092 BC00092 VJ=20.00 PL=0
MOVL C00093 BC00093 V=166.7
REFP 3 C00094 BC00094
CALL JOB:SEARCH-R1
SET P0024 P0006
SFTON P0024
MOVL C00095 BC00095 V=166.7
REFP 3 C00096 BC00096
CALL JOB:SEARCH-R1
SET P0024 P0006
SFTON P0024
SFTOF
MOVL C00097 BC00097 V=166.7
'W7A
MOVJ C00098 BC00098 VJ=40.00
MOVJ C00099 BC00099 VJ=40.00
MOVJ C00100 BC00100 VJ=40.00
MOVJ C00101 BC00101 VJ=40.00
MOVJ C00102 BC00102 VJ=40.00
MOVJ C00103 BC00103 VJ=40.00
MOVJ C00104 BC00104 VJ=40.00
MOVJ C00105 BC00105 VJ=40.00
MOVL C00106 BC00106 V=250.0
REFP 3 C00107 BC00107
CALL JOB:SEARCH-R1
SET P0280 P0006
SFTON P0280
MOVL C00108 BC00108 V=166.7
MOVL C00109 BC00109 V=250.0
MOVL C00110 BC00110 V=166.7
REFP 3 C00111 BC00111
CALL JOB:SEARCH-R1
SET P0280 P0006
MOVL C00112 BC00112 V=166.7
SFTOF
MOVL C00113 BC00113 V=333.3
MOVL C00114 BC00114 V=166.7
REFP 3 C00115 BC00115
CALL JOB:SEARCH-R1
SET P0290 P0006
SFTON P0290
MOVL C00116 BC00116 V=166.7
REFP 3 C00117 BC00117
CALL JOB:SEARCH-R1
SET P0290 P0006
MOVL C00118 BC00118 V=166.7
'DOKONCZYC SEARCH
'DOKONCZYC SEARCH
MOVJ C00119 BC00119 VJ=20.00
SFTOF
MOVJ C00120 BC00120 VJ=30.00
MOVJ C00121 BC00121 VJ=40.00
MOVJ C00122 BC00122 VJ=40.00
MOVJ C00123 BC00123 VJ=40.00
MOVJ C00124 BC00124 VJ=40.00
MOVJ C00125 BC00125 VJ=50.00
'W7B
MOVJ C00126 BC00126 VJ=50.00
MOVJ C00127 BC00127 VJ=50.00
MOVJ C00128 BC00128 VJ=30.00
MOVJ C00129 BC00129 VJ=20.00
MOVL C00130 BC00130 V=166.7
REFP 3 C00131 BC00131
CALL JOB:SEARCH-R1
SET P0281 P0006
MOVL C00132 BC00132 V=166.7
SFTON P0281
MOVL C00133 BC00133 V=166.7
MOVL C00134 BC00134 V=166.7
REFP 3 C00135 BC00135
CALL JOB:SEARCH-R1
SET P0281 P0006
MOVJ C00136 BC00136 VJ=15.00
SFTOF
MOVJ C00137 BC00137 VJ=20.00
MOVL C00138 BC00138 V=166.7
REFP 3 C00139 BC00139
CALL JOB:SEARCH-R1
SET P0291 P0006
MOVL C00140 BC00140 V=166.7
MOVL C00141 BC00141 V=166.7
REFP 3 C00142 BC00142
CALL JOB:SEARCH-R1
SET P0291 P0006
MOVL C00143 BC00143 V=166.7
MOVJ C00144 BC00144 VJ=30.00
MOVJ C00145 BC00145 VJ=30.00
MOVJ C00146 BC00146 VJ=50.00
MOVJ C00147 BC00147 VJ=50.00
'------------------------
'------------------------
'PRAWA STRONA PROFIL GORA
'------------------------
'------------------------
MOVJ C00148 BC00148 VJ=50.00
MOVJ C00149 BC00149 VJ=50.00
MOVJ C00150 BC00150 VJ=50.00
MOVJ C00151 BC00151 VJ=20.00
MOVJ C00152 BC00152 VJ=50.00
'------------------------
'W14A L
'------------------------
SFTOF
MOVJ C00153 BC00153 VJ=50.00
'------------------------
'W14A P
'------------------------
SFTOF
MOVJ C00154 BC00154 VJ=50.00
MOVJ C00155 BC00155 VJ=50.00
MOVL C00156 BC00156 V=166.7 PL=0
REFP 3 C00157 BC00157
CALL JOB:SEARCH-R1
SET P0301 P0006
SFTON P0301
MOVL C00158 BC00158 V=166.7 PL=0
REFP 3 C00159 BC00159
CALL JOB:SEARCH-R1
SET P0301 P0006
SFTON P0301
MOVL C00160 BC00160 V=166.7 PL=0
SFTOF
'------------------------
'W19A L
'------------------------
SFTOF
MOVJ C00161 BC00161 VJ=50.00
MOVL C00162 BC00162 V=200.0 PL=0
REFP 3 C00163 BC00163
CALL JOB:SEARCH-R1
SET P0302 P0006
SFTON P0302
MOVL C00164 BC00164 V=166.7 PL=0
REFP 3 C00165 BC00165
CALL JOB:SEARCH-R1
SET P0302 P0006
SFTON P0302
MOVL C00166 BC00166 V=250.0 PL=0
SFTOF
'------------------------
'W19A P
'------------------------
SFTOF
MOVJ C00167 BC00167 VJ=50.00
MOVL C00168 BC00168 V=166.7 PL=0
REFP 3 C00169 BC00169
CALL JOB:SEARCH-R1
SET P0303 P0006
SFTON P0303
MOVL C00170 BC00170 V=166.7 PL=0
REFP 3 C00171 BC00171
CALL JOB:SEARCH-R1
SET P0303 P0006
SFTON P0303
MOVL C00172 BC00172 V=166.7 PL=0
SFTOF
'------------------------
'W13A L
'------------------------
SFTOF
MOVJ C00173 BC00173 VJ=50.00
MOVL C00174 BC00174 V=166.7 PL=0
REFP 3 C00175 BC00175
CALL JOB:SEARCH-R1
SET P0304 P0006
SFTON P0304
MOVL C00176 BC00176 V=166.7 PL=0
REFP 3 C00177 BC00177
CALL JOB:SEARCH-R1
SET P0304 P0006
SFTON P0304
MOVL C00178 BC00178 V=166.7 PL=0
SFTOF
'------------------------
'W13A P
'------------------------
SFTOF
MOVJ C00179 BC00179 VJ=50.00
MOVL C00180 BC00180 V=200.0 PL=0
REFP 3 C00181 BC00181
CALL JOB:SEARCH-R1
SET P0305 P0006
SFTON P0305
MOVL C00182 BC00182 V=166.7 PL=0
REFP 3 C00183 BC00183
CALL JOB:SEARCH-R1
SET P0305 P0006
SFTON P0305
MOVL C00184 BC00184 V=250.0 PL=0
SFTOF
'------------------------
'W18A L
'------------------------
SFTOF
MOVJ C00185 BC00185 VJ=50.00
MOVL C00186 BC00186 V=200.0 PL=0
REFP 3 C00187 BC00187
CALL JOB:SEARCH-R1
SET P0306 P0006
SFTON P0306
MOVL C00188 BC00188 V=166.7 PL=0
REFP 3 C00189 BC00189
CALL JOB:SEARCH-R1
SET P0306 P0006
SFTON P0306
MOVL C00190 BC00190 V=166.7 PL=0
SFTOF
'------------------------
'W18A P
'------------------------
SFTOF
MOVJ C00191 BC00191 VJ=50.00
MOVL C00192 BC00192 V=200.0 PL=0
REFP 3 C00193 BC00193
CALL JOB:SEARCH-R1
SET P0307 P0006
SFTON P0307
MOVL C00194 BC00194 V=166.7 PL=0
REFP 3 C00195 BC00195
CALL JOB:SEARCH-R1
SET P0307 P0006
SFTON P0307
MOVL C00196 BC00196 V=166.7 PL=0
SFTOF
'------------------------
'W15A L
'------------------------
SFTOF
MOVJ C00197 BC00197 VJ=50.00
MOVL C00198 BC00198 V=200.0 PL=0
REFP 3 C00199 BC00199
CALL JOB:SEARCH-R1
SET P0308 P0006
SFTON P0308
MOVL C00200 BC00200 V=166.7 PL=0
REFP 3 C00201 BC00201
CALL JOB:SEARCH-R1
SET P0308 P0006
SFTON P0308
MOVL C00202 BC00202 V=166.7 PL=0
SFTOF
'------------------------
'W15A P
'------------------------
SFTOF
MOVJ C00203 BC00203 VJ=50.00
MOVL C00204 BC00204 V=166.7 PL=0
REFP 3 C00205 BC00205
CALL JOB:SEARCH-R1
SET P0309 P0006
SFTON P0309
MOVL C00206 BC00206 V=166.7 PL=0
REFP 3 C00207 BC00207
CALL JOB:SEARCH-R1
SET P0309 P0006
SFTON P0309
MOVL C00208 BC00208 V=166.7 PL=0
SFTOF
MOVL C00209 BC00209 V=333.3
'------------------------
'W17A L
'------------------------
MOVL C00210 BC00210 V=500.0
SFTOF
MOVJ C00211 BC00211 VJ=20.00
MOVL C00212 BC00212 V=166.7 PL=0
REFP 3 C00213 BC00213
CALL JOB:SEARCH-R1
SET P0310 P0006
SFTON P0310
MOVL C00214 BC00214 V=166.7 PL=0
REFP 3 C00215 BC00215
CALL JOB:SEARCH-R1
SET P0310 P0006
SFTON P0310
MOVL C00216 BC00216 V=166.7 PL=0
SFTOF
'------------------------
'W17A P
'------------------------
SFTOF
MOVL C00217 BC00217 V=416.7
MOVL C00218 BC00218 V=166.7 PL=0
REFP 3 C00219 BC00219
CALL JOB:SEARCH-R1
SET P0311 P0006
SFTON P0311
MOVL C00220 BC00220 V=166.7 PL=0
REFP 3 C00221 BC00221
CALL JOB:SEARCH-R1
SET P0311 P0006
SFTON P0311
MOVL C00222 BC00222 V=166.7 PL=0
SFTOF
MOVJ C00223 BC00223 VJ=10.00
MOVJ C00224 BC00224 VJ=20.00
MOVJ C00225 BC00225 VJ=50.00
MOVJ C00226 BC00226 VJ=50.00
MOVJ C00227 BC00227 VJ=70.00
MOVJ C00228 BC00228 VJ=30.00
MOVJ C00229 BC00229 VJ=30.00
'------------------------
'------------------------
'LEWA STRONA PROFIL GORA
'------------------------
'------------------------
MOVJ C00230 BC00230 VJ=30.00
MOVJ C00231 BC00231 VJ=30.00
MOVJ C00232 BC00232 VJ=30.00
'------------------------
'W17B L
'------------------------
SFTOF
MOVJ C00233 BC00233 VJ=15.00
MOVL C00234 BC00234 V=166.7 PL=0
REFP 3 C00235 BC00235
CALL JOB:SEARCH-R1
SET P0350 P0006
SFTON P0350
MOVL C00236 BC00236 V=166.7 PL=0
REFP 3 C00237 BC00237
CALL JOB:SEARCH-R1
SET P0350 P0006
SFTON P0350
MOVL C00238 BC00238 V=166.7 PL=0
SFTOF
'------------------------
'W17B P
'------------------------
SFTOF
MOVL C00239 BC00239 V=333.3
MOVL C00240 BC00240 V=166.7 PL=0
REFP 3 C00241 BC00241
CALL JOB:SEARCH-R1
SET P0351 P0006
SFTON P0351
MOVL C00242 BC00242 V=166.7 PL=0
REFP 3 C00243 BC00243
CALL JOB:SEARCH-R1
SET P0351 P0006
SFTON P0351
MOVL C00244 BC00244 V=166.7 PL=0
SFTOF
'POPRAWID DOJAZD
'------------------------
'W15B L
'------------------------
SFTOF
MOVJ C00245 BC00245 VJ=10.00
MOVL C00246 BC00246 V=166.7 PL=0
REFP 3 C00247 BC00247
CALL JOB:SEARCH-R1
SET P0352 P0006
SFTON P0352
MOVL C00248 BC00248 V=166.7 PL=0
REFP 3 C00249 BC00249
CALL JOB:SEARCH-R1
SET P0352 P0006
SFTON P0352
MOVL C00250 BC00250 V=166.7 PL=0
SFTOF
'------------------------
'W15B P
'------------------------
SFTOF
MOVJ C00251 BC00251 VJ=20.00
MOVL C00252 BC00252 V=166.7 PL=0
REFP 3 C00253 BC00253
CALL JOB:SEARCH-R1
SET P0353 P0006
SFTON P0353
MOVL C00254 BC00254 V=166.7 PL=0
REFP 3 C00255 BC00255
CALL JOB:SEARCH-R1
SET P0353 P0006
SFTON P0353
MOVL C00256 BC00256 V=166.7 PL=0
SFTOF
'------------------------
'W18B L
'------------------------
SFTOF
MOVJ C00257 BC00257 VJ=50.00
MOVL C00258 BC00258 V=166.7 PL=0
REFP 3 C00259 BC00259
CALL JOB:SEARCH-R1
SET P0354 P0006
SFTON P0354
MOVL C00260 BC00260 V=166.7 PL=0
REFP 3 C00261 BC00261
CALL JOB:SEARCH-R1
SET P0354 P0006
SFTON P0354
MOVL C00262 BC00262 V=166.7 PL=0
SFTOF
'------------------------
'W18B P
'------------------------
SFTOF
MOVJ C00263 BC00263 VJ=50.00
MOVL C00264 BC00264 V=166.7 PL=0
REFP 3 C00265 BC00265
CALL JOB:SEARCH-R1
SET P0355 P0006
SFTON P0355
MOVL C00266 BC00266 V=166.7 PL=0
REFP 3 C00267 BC00267
CALL JOB:SEARCH-R1
SET P0355 P0006
SFTON P0355
MOVL C00268 BC00268 V=166.7 PL=0
SFTOF
'------------------------
'W13B L
'------------------------
SFTOF
MOVJ C00269 BC00269 VJ=50.00
MOVL C00270 BC00270 V=166.7 PL=0
REFP 3 C00271 BC00271
CALL JOB:SEARCH-R1
SET P0356 P0006
SFTON P0356
MOVL C00272 BC00272 V=166.7 PL=0
REFP 3 C00273 BC00273
CALL JOB:SEARCH-R1
SET P0356 P0006
SFTON P0356
MOVL C00274 BC00274 V=166.7 PL=0
SFTOF
'------------------------
'W13B P
'------------------------
SFTOF
MOVJ C00275 BC00275 VJ=50.00
MOVL C00276 BC00276 V=166.7 PL=0
REFP 3 C00277 BC00277
CALL JOB:SEARCH-R1
SET P0357 P0006
SFTON P0357
MOVL C00278 BC00278 V=166.7 PL=0
REFP 3 C00279 BC00279
CALL JOB:SEARCH-R1
SET P0357 P0006
SFTON P0357
MOVL C00280 BC00280 V=166.7 PL=0
SFTOF
'------------------------
'W19B L
'------------------------
SFTOF
MOVJ C00281 BC00281 VJ=50.00
MOVL C00282 BC00282 V=166.7 PL=0
REFP 3 C00283 BC00283
CALL JOB:SEARCH-R1
SET P0358 P0006
SFTON P0358
MOVL C00284 BC00284 V=166.7 PL=0
REFP 3 C00285 BC00285
CALL JOB:SEARCH-R1
SET P0358 P0006
SFTON P0358
MOVL C00286 BC00286 V=166.7 PL=0
SFTOF
'------------------------
'W19B P
'------------------------
SFTOF
MOVJ C00287 BC00287 VJ=50.00
MOVL C00288 BC00288 V=166.7 PL=0
REFP 3 C00289 BC00289
CALL JOB:SEARCH-R1
SET P0359 P0006
SFTON P0359
MOVL C00290 BC00290 V=166.7 PL=0
REFP 3 C00291 BC00291
CALL JOB:SEARCH-R1
SET P0359 P0006
SFTON P0359
MOVL C00292 BC00292 V=166.7 PL=0
SFTOF
'------------------------
'W14B L
'------------------------
SFTOF
MOVJ C00293 BC00293 VJ=50.00
MOVL C00294 BC00294 V=166.7 PL=0
REFP 3 C00295 BC00295
CALL JOB:SEARCH-R1
SET P0360 P0006
SFTON P0360
MOVL C00296 BC00296 V=166.7 PL=0
REFP 3 C00297 BC00297
CALL JOB:SEARCH-R1
SET P0360 P0006
SFTON P0360
MOVL C00298 BC00298 V=166.7 PL=0
SFTOF
'------------------------
'W14B P
'------------------------
SFTOF
SFTOF
MOVJ C00299 BC00299 VJ=50.00
MOVJ C00300 BC00300 VJ=50.00
MOVJ C00301 BC00301 VJ=40.00
MOVL C00302 BC00302 V=166.7
SFTON P0105
MOVL C00303 BC00303 V=166.7
MACRO1 MJ#(0) ARGF24
ARCON
SFTON P0104
MOVL C00304 BC00304 V=11.3
MOVL C00305 BC00305 V=11.3
ARCOF
SFTOF
MOVL C00306 BC00306 V=333.3
MOVJ C00307 BC00307 VJ=20.00
MOVJ C00308 BC00308 VJ=30.00
COMM MOVJ C00309 BC00309 VJ=50.00
COMM MOVJ C00310 BC00310 VJ=40.00
COMM MOVJ C00311 BC00311 VJ=20.00
COMM '**********************
COMM 'W2
COMM '**********************
COMM MOVL C00312 BC00312 V=166.7
COMM SFTON P0109
COMM MOVL C00313 BC00313 V=333.3
COMM ARCON
COMM SFTON P0108
COMM MOVL C00314 BC00314 V=10.8
COMM ARCOF
COMM SFTOF
COMM MOVL C00315 BC00315 V=333.3
COMM MOVJ C00316 BC00316 VJ=40.00
MOVJ C00317 BC00317 VJ=70.00
MOVJ C00318 BC00318 VJ=30.00
MOVJ C00319 BC00319 VJ=20.00
MOVL C00320 BC00320 V=666.7
'**********************
'W3
'**********************
SFTON P0101
MOVL C00321 BC00321 V=166.7
ARCON
SFTON P0100
MOVL C00322 BC00322 V=11.7
ARCOF
MOVL C00323 BC00323 V=166.7
SFTOF
'**********************
'SPOINA_PODLOGA_BRAK_ROZP
'**********************
MOVL C00324 BC00324 V=333.3
SFTON P0099
MOVL C00325 BC00325 V=166.7
ARCON
SFTON P0098
MOVL C00326 BC00326 V=11.7
ARCOF
MOVL C00327 BC00327 V=166.7
SFTOF
'SPOINA_PODLOGA_BRAK_ROZP
MOVJ C00328 BC00328 VJ=30.00
MOVJ C00329 BC00329 VJ=30.00
MOVJ C00330 BC00330 VJ=50.00
MOVJ C00331 BC00331 VJ=30.00
MOVJ C00332 BC00332 VJ=30.00
'**********************
'W5
'**********************
MOVJ C00333 BC00333 VJ=50.00
MOVJ C00334 BC00334 VJ=50.00
MOVJ C00335 BC00335 VJ=25.00
MOVJ C00336 BC00336 VJ=30.00
'**********************
'W5
MOVL C00337 BC00337 V=333.3
'**********************
MACRO1 MJ#(0) ARGF9
SFTON P0024
MOVL C00338 BC00338 V=166.7
ARCON
WVON WEV#(2)
SFTON P0021
MOVL C00339 BC00339 V=10.8
ARCOF
WVOF
SFTOF
MOVJ C00340 BC00340 VJ=20.00
MOVJ C00341 BC00341 VJ=20.00
'**********************
'W6
'**********************
MACRO1 MJ#(0) ARGF9
SFTON P0023
MOVL C00342 BC00342 V=250.0
ARCON
WVON WEV#(2)
SFTON P0022
MOVL C00343 BC00343 V=10.8
ARCOF
WVOF
SFTOF
MOVJ C00344 BC00344 VJ=10.00
MOVJ C00345 BC00345 VJ=30.00
MOVJ C00346 BC00346 VJ=40.00
MOVJ C00347 BC00347 VJ=40.00
MOVJ C00348 BC00348 VJ=40.00
MOVJ C00349 BC00349 VJ=40.00
MOVJ C00350 BC00350 VJ=20.00
MOVJ C00351 BC00351 VJ=10.00
MOVJ C00352 BC00352 VJ=20.00
MOVL C00353 BC00353 V=166.7
MACRO1 MJ#(0) ARGF14
MOVL C00354 BC00354 V=166.7
SFTON P0280
MOVL C00355 BC00355 V=166.7 PL=0
ARCON ASF#(22)
MOVL C00356 BC00356 V=9.2
MOVL C00357 BC00357 V=9.2
SFTON P0290
MOVL C00358 BC00358 V=9.2
MOVL C00359 BC00359 V=9.2
ARCOF
SFTOF
MOVL C00360 BC00360 V=250.0
MOVL C00361 BC00361 V=416.7
MOVJ C00362 BC00362 VJ=30.00
MOVJ C00363 BC00363 VJ=30.00
MOVJ C00364 BC00364 VJ=30.00
MOVJ C00365 BC00365 VJ=30.00
MOVJ C00366 BC00366 VJ=30.00
'7b
MOVL C00367 BC00367 V=333.3
MOVL C00368 BC00368 V=333.3
SFTON P0281
MOVL C00369 BC00369 V=166.7 PL=0
ARCON ASF#(22)
MOVL C00370 BC00370 V=9.2
MOVL C00371 BC00371 V=9.2
SFTON P0291
MOVL C00372 BC00372 V=9.2
MOVL C00373 BC00373 V=9.2
MOVL C00374 BC00374 V=9.2
ARCOF
SFTOF
'TUTAJ DODAC 7
'TUTAJ DODAC 7
'TUTAJ DODAC 7
MOVL C00375 BC00375 V=333.3
MOVL C00376 BC00376 V=333.3
MOVL C00377 BC00377 V=333.3
MOVJ C00378 BC00378 VJ=20.00
MOVJ C00379 BC00379 VJ=30.00
MOVJ C00380 BC00380 VJ=50.00
MOVJ C00381 BC00381 VJ=50.00
'**********************
'W9
'**********************
MACRO1 MJ#(0) ARGF24
SFTON P0103
MOVL C00382 BC00382 V=250.0
ARCON
SFTON P0102
MOVL C00383 BC00383 V=10.8
ARCOF
SFTOF
MOVL C00384 BC00384 V=333.3
MOVJ C00385 BC00385 VJ=50.00
MOVJ C00386 BC00386 VJ=70.00
MOVJ C00387 BC00387 VJ=50.00
MOVJ C00388 BC00388 VJ=20.00
'**********************
'W10
'**********************
SFTON P0107
MOVL C00389 BC00389 V=250.0
ARCON
SFTON P0106
MOVL C00390 BC00390 V=11.3
ARCOF
SFTOF
MOVL C00391 BC00391 V=333.3
MOVJ C00392 BC00392 VJ=50.00
MOVJ C00393 BC00393 VJ=50.00
'**********************
'**********************
'POCZATEK SPAWANIA BOKI
'**********************
'**********************
MOVJ C00394 BC00394 VJ=50.00
MOVJ C00395 BC00395 VJ=50.00
'**********************
'W13A
'**********************
SFTON P0305
MOVL C00396 BC00396 V=250.0 PL=0
SFTOF
MACRO1 MJ#(0) ARGF10
ARCON
SFTON P0304
MOVL C00397 BC00397 V=10.8
ARCOF
SFTOF
MOVL C00398 BC00398 V=250.0
'W13B
MOVJ C00399 BC00399 VJ=30.00
MOVJ C00400 BC00400 VJ=50.00
MOVL C00401 BC00401 V=500.0
'**********************
'W13B
'**********************
SFTON P0356
MOVL C00402 BC00402 V=166.7 PL=0
SFTOF
ARCON
SFTON P0357
MOVL C00403 BC00403 V=10.8
ARCOF
SFTOF
MOVL C00404 BC00404 V=250.0
MOVJ C00405 BC00405 VJ=30.00
COMM MOVJ C00406 BC00406 VJ=40.00
COMM MOVJ C00407 BC00407 VJ=30.00
COMM MOVJ C00408 BC00408 VJ=30.00
COMM '**********************
COMM 'W14A
COMM '**********************
COMM MOVL C00409 BC00409 V=250.0
COMM SFTON P0301
COMM MOVL C00410 BC00410 V=133.3 PL=0
COMM SFTOF
COMM ARCON
COMM SFTON P0301
COMM MOVL C00411 BC00411 V=10.8
COMM ARCOF
COMM SFTOF
COMM MOVL C00412 BC00412 V=150.0
COMM MOVJ C00413 BC00413 VJ=40.00
COMM MOVJ C00414 BC00414 VJ=30.00
COMM MOVJ C00415 BC00415 VJ=30.00
COMM MOVJ C00416 BC00416 VJ=30.00
COMM MOVJ C00417 BC00417 VJ=30.00
COMM '**********************
COMM 'W14B
COMM '**********************
COMM SFTON P0360
COMM MOVL C00418 BC00418 V=333.3
COMM MOVL C00419 BC00419 V=166.7 PL=0
COMM ARCON
COMM MOVL C00420 BC00420 V=10.8
COMM ARCOF
COMM SFTOF
COMM MOVL C00421 BC00421 V=250.0
COMM MOVJ C00422 BC00422 VJ=40.00
COMM MOVJ C00423 BC00423 VJ=40.00
COMM MOVJ C00424 BC00424 VJ=30.00
MOVJ C00425 BC00425 VJ=40.00
MOVJ C00426 BC00426 VJ=30.00
MOVJ C00427 BC00427 VJ=30.00
MOVJ C00428 BC00428 VJ=30.00
MOVJ C00429 BC00429 VJ=30.00
MOVJ C00430 BC00430 VJ=30.00
'**********************
'W15A
'**********************
SFTON P0309
MOVL C00431 BC00431 V=166.7
MOVL C00432 BC00432 V=166.7 PL=0
SFTOF
ARCON
SFTON P0308
MOVL C00433 BC00433 V=10.8
ARCOF
SFTOF
MOVL C00434 BC00434 V=150.0
MOVJ C00435 BC00435 VJ=30.00
MOVJ C00436 BC00436 VJ=50.00
MOVJ C00437 BC00437 VJ=50.00
MOVJ C00438 BC00438 VJ=50.00
MOVJ C00439 BC00439 VJ=50.00
MOVJ C00440 BC00440 VJ=50.00
'**********************
'W15B
'**********************
SFTON P0352
MOVL C00441 BC00441 V=250.0
MOVL C00442 BC00442 V=83.3 PL=0
SFTOF
ARCON
SFTON P0353
MOVL C00443 BC00443 V=10.8
ARCOF
MOVL C00444 BC00444 V=66.7
SFTOF
MOVJ C00445 BC00445 VJ=40.00
MOVJ C00446 BC00446 VJ=50.00
MOVJ C00447 BC00447 VJ=50.00
'BRAK W TEJ DLUGOSCI
'**********************
'W16A
'**********************
'**********************
'W16B
'**********************
'BRAK W TEJ DLUGOSCI
'**********************
'W17A
'**********************
MOVJ C00448 BC00448 VJ=50.00
MOVJ C00449 BC00449 VJ=50.00
'**********************
'W17A
'**********************
SFTON P0310
MOVL C00450 BC00450 V=333.3
MOVL C00451 BC00451 V=166.7 PL=0
SFTOF
ARCON
SFTON P0311
MOVL C00452 BC00452 V=10.8
ARCOF
SFTOF
MOVL C00453 BC00453 V=333.3
MOVJ C00454 BC00454 VJ=30.00
MOVJ C00455 BC00455 VJ=30.00
MOVJ C00456 BC00456 VJ=50.00
MOVJ C00457 BC00457 VJ=50.00
MOVJ C00458 BC00458 VJ=50.00
MOVJ C00459 BC00459 VJ=50.00
MOVJ C00460 BC00460 VJ=50.00
MOVJ C00461 BC00461 VJ=30.00
MOVJ C00462 BC00462 VJ=30.00
'**********************
'W17B
'**********************
SFTON P0351
MOVL C00463 BC00463 V=166.7
MOVL C00464 BC00464 V=166.7 PL=0
SFTOF
ARCON
SFTON P0350
MOVL C00465 BC00465 V=10.8
ARCOF
SFTOF
MOVL C00466 BC00466 V=250.0
MOVJ C00467 BC00467 VJ=30.00
MOVJ C00468 BC00468 VJ=30.00
MOVJ C00469 BC00469 VJ=30.00
MOVJ C00470 BC00470 VJ=30.00
MOVJ C00471 BC00471 VJ=40.00
'**********************
'W18A
'**********************
SFTON P0306
MOVL C00472 BC00472 V=333.3
MOVL C00473 BC00473 V=166.7 PL=0
SFTOF
ARCON
SFTON P0307
MOVL C00474 BC00474 V=10.8
ARCOF
SFTOF
MOVL C00475 BC00475 V=250.0
MOVJ C00476 BC00476 VJ=30.00
MOVJ C00477 BC00477 VJ=30.00
MOVJ C00478 BC00478 VJ=50.00
MOVJ C00479 BC00479 VJ=50.00
MOVJ C00480 BC00480 VJ=50.00
'**********************
'W18B
'**********************
SFTON P0355
MOVL C00481 BC00481 V=166.7
MOVL C00482 BC00482 V=166.7 PL=0
SFTOF
ARCON
SFTON P0354
MOVL C00483 BC00483 V=10.8
ARCOF
MOVL C00484 BC00484 V=250.0
SFTOF
MOVJ C00485 BC00485 VJ=30.00
MOVJ C00486 BC00486 VJ=30.00
MOVJ C00487 BC00487 VJ=40.00
MOVJ C00488 BC00488 VJ=50.00
MOVJ C00489 BC00489 VJ=30.00
'**********************
'W19A
'**********************
MOVL C00490 BC00490 V=166.7
SFTON P0303
MOVL C00491 BC00491 V=166.7 PL=0
SFTOF
ARCON
SFTON P0302
MOVL C00492 BC00492 V=10.8
ARCOF
SFTOF
MOVL C00493 BC00493 V=150.0
MOVJ C00494 BC00494 VJ=30.00
MOVJ C00495 BC00495 VJ=50.00
MOVJ C00496 BC00496 VJ=50.00
'**********************
'W19B
'**********************
SFTON P0358
MOVL C00497 BC00497 V=500.0
MOVL C00498 BC00498 V=166.7 PL=0
SFTOF
ARCON
SFTON P0359
MOVL C00499 BC00499 V=10.8
ARCOF
SFTOF
MOVL C00500 BC00500 V=250.0
MOVJ C00501 BC00501 VJ=40.00
MOVJ C00502 BC00502 VJ=50.00
CALL JOB:MOVE_OUT_OF_TUNNEL
END
